// TIA Portal V16 export
// export: Created 2024-02-03T21:03:34.0471067Z, ExportSetting WithDefaults, DisplayName Totally Integrated Automation Portal, DisplayVersion V16 Update 6, DisplayName TIA Portal Version Control Interface, DisplayVersion V16 Update 2, DisplayName TIA Portal Openness, DisplayVersion V16 Update 6, DisplayName SINAMICS Startdrive Advanced, DisplayVersion V16 Update 5, DisplayName SINAMICS Startdrive G130, G150, S120, S150, SINAMICS MV, S210, DisplayVersion V16 Update 5, DisplayName SINAMICS Startdrive G110M, G120, G120C, G120D, G120P, G115D, DisplayVersion V16 Update 5, DisplayName STEP 7 Professional, DisplayVersion V16 Update 6, DisplayName STEP 7 Safety, DisplayVersion V16, DisplayName WinCC Professional, DisplayVersion V16 Update 6
DATA_BLOCK "test_blocks_DB"   // DB5
VERSION : 0.1
// stored: AutoNumber true, DBAccessibleFromOPCUA true, InstanceOfName test_blocks, InstanceOfType FB
"test_blocks"
   // VAR
   //    MC_POWER_Instance { S7_SetPoint := 'True'} : MC_POWER;
   //    MC_RESET_Instance { S7_SetPoint := 'True'} : MC_RESET;
   //    MC_HOME_Instance { S7_SetPoint := 'True'} : MC_HOME;
   // END_VAR
BEGIN
END_DATA_BLOCK
